TYPE ST_NcAxisStatus :
	STRUCT
		Disabled		   : BOOL;
		SynchronizedMotion : BOOL;
		Coupled			   : BOOL;
	END_STRUCT
END_TYPE

(* stored: Version 1.1.0.1, ProductVersion 3.1.4026.20
   DUT ST_NcAxisStatus: Id {cabe5152-d2bb-44d0-b22c-22252028b977} *)
